TYPE T_SIM_ACTUATOR_STAT :
STRUCT
	bInitialised:	BOOL	:= FALSE;						(* If TRUE, power simulator is initialised *)

	nErrorCode: 	DINT 	:= E_ACTUATOR_ERROR.NOT_INITIALISED;	(* Error code *)
	sErrorText: 	STRING 	:= 'NOT INITIALISED'; 			(* Error text *)
	sStatus: 		STRING 	:= 'ERROR'; 					(* power status in textual form, e.g. 'OFF' *)
END_STRUCT
END_TYPE

(* stored: Version 1.1.0.1, ProductVersion 3.1.4024.3
   DUT T_SIM_ACTUATOR_STAT: Id {91af19d4-208f-48f7-a423-e4ef68fbafcd} *)
